{attribute 'linkalways'} 
{attribute 'no_explicit_call' := 'This FB is a CLASS and must be accessed using methods or properties'}
{attribute 'enable_dynamic_creation'}
FUNCTION_BLOCK Node_F_VN_CreateBandrejectGaussianFilter EXTENDS VisionNode
VAR
    ipFilter : _ITcVnImage;
    nWidth : _UDINT(2);
    nHeight : _UDINT(2);
    bDoublePrecision : _BOOL(FALSE);
    bOriginAtCenter : _BOOL(FALSE);
    fCutoffDistance : _LREAL(1.0);
    fBandWidth : _LREAL(1.0);
    hrPrev : _HRESULT(S_OK);
	hresult : _HRESULT(S_OK);
END_VAR

METHOD PUBLIC  Clone : I_Node
VAR
	pNode : POINTER TO Node_F_VN_CreateBandrejectGaussianFilter;
END_VAR
pNode := __NEW(Node_F_VN_CreateBandrejectGaussianFilter);
Clone := pNode^;
END_METHOD

METHOD FB_init : BOOL
VAR_INPUT
	bInitRetains : BOOL; // if TRUE, the retain variables are initialized (warm start / cold start)
	bInCopyCode : BOOL;  // if TRUE, the instance afterwards gets moved into the copy code (online change)
END_VAR
AddParameter('nWidth', nWidth);
AddParameter('nHeight', nHeight);
AddParameter('bDoublePrecision', bDoublePrecision);
AddParameter('bOriginAtCenter', bOriginAtCenter);
AddParameter('fCutoffDistance', fCutoffDistance);
AddParameter('fBandWidth', fBandWidth);
AddInput('hrPrev', hrPrev);
AddOutput('ipFilter', ipFilter);
AddOutput('hresult',hresult);
END_METHOD

METHOD PROTECTED OnExecute
hresult.Value := F_VN_CreateBandrejectGaussianFilter(
    ipFilter := ipFilter.Value,
	nWidth := nWidth.Value,
    nHeight := nHeight.Value,
    bDoublePrecision := bDoublePrecision.Value,
    bOriginAtCenter := bOriginAtCenter.Value,
    fCutoffDistance := fCutoffDistance.Value,
    fBandWidth := fBandWidth.Value,
	hrPrev:= hrPrev.Value);
END_METHOD

METHOD PUBLIC PreExecutionCheck
VAR_INPUT
	Check : I_PreExecutionChecks;
END_VAR
Check.IsTrue(nWidth.IsEven, 'nWidth must be an even number');
Check.IsTrue(nHeight.IsEven, 'nHeight must be an even number');
Check.IsTrue((nWidth.Value >= 2), 'nWidth must be greater than or equal to 2');
Check.IsTrue((nHeight.Value >= 2), 'nWidth must be greater than or equal to 2');
Check.IsTrue((fCutoffDistance.Value > 0), 'nCutoffDistance must be greater than 0');
Check.IsTrue((fBandWidth.Value > 0), 'fBandWidth must be greater than 0');
END_METHOD

END_FUNCTION_BLOCK

(* stored: Version 1.1.0.1, ProductVersion 3.1.4024.13
   POU Node_F_VN_CreateBandrejectGaussianFilter: Id {199faafd-c98c-0e4c-3910-db3e41643983}, SpecialFunc None
   Folder Constructor: Id {b29559b8-db48-098a-370f-2cea27e81901}
   Method Clone: Id {0fa621f3-7faa-0de4-3944-7ac74831ac5e}
   Method FB_init: Id {93f3107a-196b-0eaf-24e8-1dd518451164}
   Method OnExecute: Id {ae0020e3-873d-0c72-0fa8-ce67263db0db}
   Method PreExecutionCheck: Id {56c0f2da-3177-029e-164d-c0edc44da52a} *)
